# EPICS autosave request: xspdApp/Db/ADXSPD_settings.req
file "ADBase_settings.req", P=$(P),  R=$(R)
file "NDFile_settings.req", P=$(P),  R=$(R)
